FUNCTION_BLOCK WAREHOUSE
  {SET_ATTRIBUTE(OpcUa, POINT.STARTPOINT)}
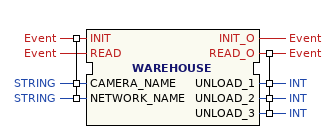
  EVENT_INPUT
    INIT WITH CAMERA_NAME, NETWORK_NAME;
    READ;
  END_EVENT
  EVENT_OUTPUT
    INIT_O;
    READ_O WITH UNLOAD_1, UNLOAD_2, UNLOAD_3;
  END_EVENT
  VAR_INPUT
    CAMERA_NAME : STRING; {SET_ATTRIBUTE(OpcUa, Variable.RUN)}
    NETWORK_NAME : STRING; {SET_ATTRIBUTE(OpcUa, Variable.RUN)}
  END_VAR
  VAR_OUTPUT
    UNLOAD_1 : INT; {SET_ATTRIBUTE(OpcUa, Variable.RUN)}
    UNLOAD_2 : INT; {SET_ATTRIBUTE(OpcUa, Variable.RUN)}
    UNLOAD_3 : INT; {SET_ATTRIBUTE(OpcUa, Variable.RUN)}
  END_VAR
END_FUNCTION_BLOCK
